(* IEC 61131-3 sources: git_feedingMachine/app/src/StateMachine/StateObject, 7 files *)

(* ---- ErrorState.st ---- *)
USING TankLib;
USING Siemens.Simatic.S71500.MotionControl.Native;
USING Siemens.Simatic.Motion;
NAMESPACE Siemens.Simatic.StateMachine

    CLASS PUBLIC ErrorState IMPLEMENTS IState
        VAR
            _feedAxis : REF_TO PosAxis;
            _tank : REF_TO Tank;
            canGoNext : BOOL := FALSE;
        END_VAR
        //执行动作逻辑
        METHOD PUBLIC ExcuteJob
            VAR_EXTERNAL
                resetError : BOOL;
            END_VAR
            IF resetError THEN
                canGoNext := TRUE;
                _feedAxis^.ResetAxis();
            END_IF;
        END_METHOD

        //处理状态
        METHOD PUBLIC HandleState
            VAR_INPUT
                context : REF_TO FeedingMachine;
                tank : REF_TO Tank;
                feedAxis : REF_TO PosAxis;
            END_VAR
            VAR_EXTERNAL
                sinkEmptySensor : BOOL;
                axisStop : BOOL;
                powerOff : BOOL;
                tankEmptySensor : BOOL;
            END_VAR
            THIS._tank := tank;
            THIS._feedAxis := feedAxis;

            //执行Action
            THIS.ExcuteJob();

            //断电或空罐
            IF powerOff THEN
                 //切换到OFFState状态对象
                context^.SetState(context^.GetOffState(),_tank,_feedAxis);
            END_IF;

            //等待可跳转信号
            IF canGoNext THEN
                canGoNext := FALSE;
                IF NOT _feedAxis^.GetAxisStatus().error THEN
                    //切换到StopState状态对象
                    context^.SetState(context^.GetStopState(),_tank,_feedAxis);
                END_IF;
            END_IF;
        END_METHOD

        //获取状态
        METHOD PUBLIC GetState : STRING
            GetState:='Error';
        END_METHOD

    END_CLASS

END_NAMESPACE

(* ---- FillSinkState.st ---- *)
USING TankLib;
USING Siemens.Simatic.S71500.MotionControl.Native;
USING Siemens.Simatic.Motion;
NAMESPACE Siemens.Simatic.StateMachine

    CLASS PUBLIC FillSinkState IMPLEMENTS IState
        VAR
            _feedAxis : REF_TO PosAxis;
            _tank : REF_TO Tank;
        END_VAR

        //执行动作逻辑
        METHOD PUBLIC ExcuteJob
            _tank^.Feeding();
            _feedAxis^.DisableAxis(stopMode := 1);
        END_METHOD

        //处理状态
        METHOD PUBLIC HandleState
            VAR_INPUT
                context : REF_TO FeedingMachine;
                tank : REF_TO Tank;
                feedAxis : REF_TO PosAxis;
            END_VAR
            VAR_EXTERNAL
                sinkFullSensor:BOOL;
                powerOff : BOOL;
                tankEmptySensor : BOOL;
            END_VAR

            THIS._tank := tank;
            THIS._feedAxis := feedAxis;

            //执行Action
            THIS.ExcuteJob();

            //断电或空罐
            IF powerOff OR tankEmptySensor THEN
                //切换到OFFState状态对象
                context^.SetState(context^.GetOffState(),_tank,_feedAxis);
            END_IF;

            //等待可跳转信号
            IF sinkFullSensor THEN
                //切换到ReadyState状态对象
                context^.SetState(context^.GetReadyState(),_tank,_feedAxis);
            END_IF;
        END_METHOD

        //获取状态
        METHOD PUBLIC GetState : STRING
            GetState:='Filling Sink';
        END_METHOD

    END_CLASS

END_NAMESPACE

(* ---- FillTankState.st ---- *)
USING TankLib;
USING Siemens.Simatic.S71500.MotionControl.Native;
USING Siemens.Simatic.Motion;
NAMESPACE Siemens.Simatic.StateMachine

    CLASS PUBLIC FillTankState IMPLEMENTS IState
        VAR
            _feedAxis : REF_TO PosAxis;
            _tank : REF_TO Tank;
        END_VAR

        //执行动作逻辑
        METHOD Public ExcuteJob
            _tank^.Filling();
            _feedAxis^.DisableAxis(stopMode := 1);
        END_METHOD

        //处理状态
        METHOD PUBLIC HandleState
            VAR_INPUT
                context : REF_TO FeedingMachine;
                tank : REF_TO Tank;
                feedAxis : REF_TO PosAxis;
            END_VAR
            VAR_EXTERNAL
                tankFullSensor :BOOL;
                powerOff : BOOL;
                tankEmptySensor : BOOL;
            END_VAR

            THIS._tank := tank;
            THIS._feedAxis := feedAxis;

            //执行Action
            THIS.ExcuteJob();

            //断电或空罐
            IF powerOff OR tankEmptySensor THEN
                //切换到OFFState状态对象
                context^.SetState(context^.GetOffState(),_tank,_feedAxis);

            END_IF;
            //等待可跳转信号
            IF tankFullSensor THEN
                //切换到fILLSinkState状态对象
                context^.SetState(context^.GetFillSinkState(),_tank,_feedAxis);
            END_IF;
        END_METHOD

        //获取状态
        METHOD PUBLIC GetState : STRING
            GetState:='Filling Tank';
        END_METHOD

    END_CLASS

END_NAMESPACE

(* ---- OffState.st ---- *)
USING TankLib;
USING Siemens.Simatic.S71500.MotionControl.Native;
USING Siemens.Simatic.Motion;

NAMESPACE Siemens.Simatic.StateMachine

    CLASS PUBLIC OffState IMPLEMENTS IState
        VAR
            _feedAxis : REF_TO PosAxis;
            _tank: REF_TO Tank;
        END_VAR

        //执行动作逻辑
        METHOD PUBLIC ExcuteJob
            _tank^.Close();
            _feedAxis^.ResetCmds();
            _feedAxis^.DisableAxis(stopMode := 1);
        END_METHOD

        //处理状态
        METHOD PUBLIC HandleState
            VAR_INPUT
                context : REF_TO FeedingMachine;
                tank : REF_TO Tank;
                feedAxis : REF_TO PosAxis;
            END_VAR
            VAR_EXTERNAL
                powerOn :BOOL;
                powerOff : BOOL;
            END_VAR

            THIS._tank := tank;
            THIS._feedAxis := feedAxis;

            //执行Action
            THIS.ExcuteJob();

            //等待可跳转信号
            IF powerOn AND NOT(powerOff) THEN
                //切换到FillSink状态对象
                context^.SetState(context^.GetFillTankState(),_tank,_feedAxis);
            END_IF;
        END_METHOD

        //获取状态
        METHOD PUBLIC GetState : STRING
            GetState:='OFF';
        END_METHOD

    END_CLASS

END_NAMESPACE

(* ---- ReadyState.st ---- *)
USING TankLib;
USING Siemens.Simatic.S71500.MotionControl.Native;
USING Siemens.Simatic.Motion;
NAMESPACE Siemens.Simatic.StateMachine

    CLASS PUBLIC ReadyState IMPLEMENTS IState
        VAR
            _feedAxis : REF_TO PosAxis;
            _tank : REF_TO Tank;
            canGoNext : BOOL := FALSE;
        END_VAR

        //执行动作逻辑
        METHOD PUBLIC ExcuteJob
            VAR_EXTERNAL
                axisStart : BOOL;
                errorID : WORD;
            END_VAR
            _tank^.close();
            IF axisStart THEN
                _feedAxis^.EnableAxis(startmode := 1);
                _feedAxis^.HomeAxis(position := 0.0, homingMode := 0);
                canGoNext:=TRUE;
            END_IF;
        END_METHOD

        //处理状态
        METHOD PUBLIC HandleState
            VAR_INPUT
                context : REF_TO FeedingMachine;
                tank : REF_TO Tank;
                feedAxis : REF_TO PosAxis;
            END_VAR
            VAR_EXTERNAL
                powerOff : BOOL;
                tankEmptySensor : BOOL;
                errorID : WORD;
                sinkEmptySensor:Bool;
            END_VAR

            THIS._tank := tank;
            THIS._feedAxis := feedAxis;

            //执行Action
            THIS.ExcuteJob();
            //轴控错误
            IF _feedAxis^.GetAxisStatus().Error THEN
                //切换到Error状态对象
                context^.SetState(context^.GetErrorState(),_tank,_feedAxis);;
            END_IF;

            //断电或空罐
            IF powerOff OR tankEmptySensor THEN
                 //切换到OFFState状态对象
                context^.SetState(context^.GetOffState(),_tank,_feedAxis);
            END_IF;

            //等待可跳转信号
            IF canGoNext AND NOT(sinkEmptySensor) AND _feedAxis^.GetAxisStatus().enabled AND _feedAxis^.GetAxisStatus().homed THEN
                canGoNext:=FALSE;
                //切换到RunState状态对象
                context^.SetState(context^.GetRunState(),_tank,_feedAxis);
            END_IF;
        END_METHOD

        //获取状态
        METHOD PUBLIC GetState : STRING
            GetState:='Ready';
        END_METHOD

    END_CLASS

END_NAMESPACE

(* ---- RunState.st ---- *)
USING TankLib;
USING Siemens.Simatic.S71500.MotionControl.Native;
USING Siemens.Simatic.Motion;

NAMESPACE Siemens.Simatic.StateMachine

    CLASS PUBLIC RunState IMPLEMENTS IState
        VAR
            _feedAxis : REF_TO PosAxis;
            _tank: REF_TO Tank;
        END_VAR

        //执行动作逻辑
        METHOD PUBLIC ExcuteJob
            // VAR
            //     AxMoveCmd:itfCommand;
            // END_VAR
            VAR_EXTERNAL
                errorID : WORD;
            END_VAR
            _feedAxis^.PosAbsolute(position := 4000.0,velocity := 50.0,acceleration := -1.0,deceleration := -1.0);
        END_METHOD

        //处理状态
        METHOD PUBLIC HandleState
            VAR_INPUT
                context : REF_TO FeedingMachine;
                tank : REF_TO Tank;
                feedAxis : REF_TO PosAxis;
            END_VAR
            VAR_EXTERNAL
                axisStop:BOOL;
                sinkEmptySensor : BOOL;
                powerOff : BOOL;
                tankEmptySensor : BOOL;
                errorID : WORD;
            END_VAR

            THIS._tank := tank;
            THIS._feedAxis := feedAxis;

            //执行Action
            this.ExcuteJob();

            //轴控错误
            IF _feedAxis^.GetAxisStatus().Error THEN
                //切换到Error状态对象
                context^.SetState(context^.GetErrorState(),_tank,_feedAxis);;
            END_IF;

            //断电或空罐
            IF powerOff OR tankEmptySensor THEN
                 //切换到OFFState状态对象
                context^.SetState(context^.GetOffState(),_tank,_feedAxis);
            END_IF;

            //等待可跳转信号
            IF axisStop OR sinkEmptySensor THEN
                //切换到StopState状态对象
                context^.SetState(context^.GetStopState(),_tank,_feedAxis);
            END_if;
        END_METHOD

        //获取状态
        METHOD PUBLIC GetState : STRING
            GetState:='Runing';
        END_METHOD

    END_CLASS

END_NAMESPACE

(* ---- StopState.st ---- *)
USING TankLib;
USING Siemens.Simatic.S71500.MotionControl.Native;
USING Siemens.Simatic.Motion;
NAMESPACE Siemens.Simatic.StateMachine

    CLASS PUBLIC StopState IMPLEMENTS IState
        VAR
            _feedAxis : REF_TO PosAxis;
            _tank : REF_TO Tank;
        END_VAR

        //执行动作逻辑
        METHOD PUBLIC ExcuteJob
            _feedAxis^.StopAxis(deceleration := -1.0, jerk := -1.0);
        END_METHOD

        //处理状态
        METHOD PUBLIC HandleState
            VAR_INPUT
                context : REF_TO FeedingMachine;
                tank : REF_TO Tank;
                feedAxis : REF_TO PosAxis;
            END_VAR
            VAR_EXTERNAL
                axisStart : BOOL;
                axisStop : BOOL;
                powerOff : BOOL;
                tankEmptySensor : BOOL;
                errorID : WORD;
            END_VAR
            THIS._tank:=tank;
            THIS._feedAxis:=feedAxis;

            //执行Action
            THIS.ExcuteJob();

             //轴控错误
             IF _feedAxis^.GetAxisStatus().Error THEN
                //切换到Error状态对象
                context^.SetState(context^.GetErrorState(),_tank,_feedAxis);;
            END_IF;

            //断电或空罐
            IF powerOff OR tankEmptySensor THEN
                 //切换到OFFState状态对象
                context^.SetState(context^.GetOffState(),_tank,_feedAxis);
                END_IF;

            //等待可跳转信号
            IF axisStart AND NOT axisStop THEN
                //切换到FillSinkState状态对象
                context^.SetState(context^.GetFillSinkState(),_tank,_feedAxis);
            END_IF;

        END_METHOD

        //获取状态
        METHOD PUBLIC GetState : STRING
            GetState:='Stoped';
        END_METHOD

    END_CLASS

END_NAMESPACE
